(* PLC project PLC1, Beckhoff Automation GmbH TwinCAT PLC Control 3.5.13.21 *)
(* stored: creationDateTime 2023-10-09T14:50:05.3128297, modificationDateTime 2023-10-09T14:50:05.3189547 *)

PROGRAM MAIN
VAR	
	{region 'NC Variables'}
	// Status Array of MCS Position
	MCS_Positions : ARRAY[1..MAX_MCS_AXES] OF LREAL;	
	// Axis Control Ref for ACS
	ACS_Axis		: ARRAY[1..MAX_ACS_AXES] OF Axis_Ref;
	// Axis Control Ref for MCS
	MCS_Axis		: ARRAY[1..MAX_MCS_AXES] OF Axis_Ref;
	// ACS Axis Power Block
	mcACS_Power 	: ARRAY[1..MAX_ACS_AXES] OF MC_Power;
	// MCS Axis Power Block
	mcMCS_Power 	: ARRAY[1..MAX_MCS_AXES] OF MC_Power;
	// Axis Set Position Block
	mcSetPosition 	: ARRAY[1..MAX_ACS_AXES] OF MC_SetPosition;
	{endregion}
		 
	{region  'Kinematics Variables'}
	// Kinematic Model Reference
	{attribute 'TcInitSymbol'}
	oidTrafo			: OTCID;
	// Struct In from Kin Channel
	in_stKinToPlc      AT %I*     : NCTOPLC_NCICHANNEL_REF;
	// Struct Out to Kin Channel
	out_stPlcToKin     AT %Q*     : PLCTONC_NCICHANNEL_REF;	 
	// Axes Configuration Structure
	stAxesConfig		: ST_KinAxes;
	// Kinematics Configuration Group			  
	fbConfigKinGroup	: FB_KinConfigGroup;
	// Reset the Kin Group
	fbResetKinGroup   : FB_KinResetGroup;
	// Calculating the Trafo
	fbKinCalcTrafo		: FB_KinCalcTrafo;
	// Struct of position into the calculation
    stAxesPosIn			: ARRAY[1..8] OF LREAL;
	// Struct of positions out
    stAxesPosOut		: ARRAY[1..8] OF LREAL;			  
	// Scara Meta Info 
	uScaraMetaInfoIn	: U_KinMetaInfo;
	// Scara Meta Info
    uScaraMetaInfoOut	: U_KinMetaInfo;
  	// Unlock Trafo
	fbUnlockTrafoParam	: FB_KinUnlockTrafoParam;
	// Lock Trafo
	fbLockTrafoParam	: FB_KinLockTrafoParam;
	// ADS Write Block
    fbADSWRITE			: ADSWRITE;	
	// Parameter ID to Change (*Inner Arm Length*)
	pidTrafo			: UDINT := 16#05010020; 
	// Value to write to the parameter
	fParamValue			: LREAL := 400.0;			  
	{endregion}

	{region  'General System Variables'}
	// Loop Iterator
	I_itr			: INT;
	{endregion}
		 
	{region 'State Machine Variables'}
	// State of the state machine
	nState 			: INT;
	// Control Variables
	bStart, bHalt, bDoneMoving, bCalcTrafo, bAdjustTrafo, bRepeat : BOOL;
	{endregion}
END_VAR
VAR CONSTANT
	{region  'Axes Constants'}
	// ACS Axes Count
	MAX_ACS_AXES 		: INT := 4;
	// MCS Axes Count
	MAX_MCS_AXES 		: INT := 4;
	// Joint Positions
	AXES_JOINT_POSE	: ARRAY[1..MAX_ACS_AXES] OF LREAL := [0.0, 90.0, 0.0, 0.0];
	{endregion}
END_VAR

            // Simple NC State Machine

CASE nState OF
	0:	// Start the state machine
		IF bStart THEN
			bStart := FALSE;
			nState := nState + 10;
		END_IF
	
	10..40: 
		// Power on all axis (Both ACS and MCS)
		ACS_MCS_Power();
	  
	50: 
		// Step 1 - Assemble the Axes List Struct
		Step_1_Axes_List();
	 
	60..70:	
		// Step 3 - might have an issue at Step 2, so here is where you'll fix it
		Step_3_Fix_Kin_Config();
			   
	80: 
		//	Step 2 - Configure Kinematic Group
		Step_2_Configure_Kin_Group();
					  
	90: 
		(*
		** Move the robot!
		*)
		(*******************************************)	 
		// Command to move on from this step				   
		IF bDoneMoving THEN
			bDoneMoving := FALSE;
			nState := nState + 10;
		END_IF
		(*******************************************)	
		
	100: 
		// Step 5 - Break the Kinematic Group
		Step_5_Reconfig_Kin_Group(); 				   
		 
	110: 
		// Wait state before adjustment
		IF bAdjustTrafo THEN
			bAdjustTrafo := FALSE;
			nState := nState + 10;
		END_IF
	
	120..140:
		// Step 6 - Unlock Trafo and Modify Params
		Step_6_Adjust_Trafo();	 
		
	150: 
		// Check if repeating state machine
		IF bRepeat THEN
			bRepeat := FALSE;
			nState := 60;
		END_IF		
END_CASE


// Step 4 - Calculate the Transformation
IF bCalcTrafo THEN
	Step_4_Calc_Trafo();
END_IF

	 
          

ACTION Step_1_Axes_List:
                (*

// Assign the ACS Axes
FOR I_itr := 1 TO MAX_ACS_AXES DO
	stAxesConfig.nAxisIdsAcs[I_itr] := ACS_Axis[I_itr].NcToPlc.AxisId;
END_FOR
// Assign the MCS Axes
FOR I_itr := 1 TO MAX_MCS_AXES DO
	stAxesConfig.nAxisIdsMcs[I_itr] := MCS_Axis[I_itr].NcToPlc.AxisId;
END_FOR

*)


nState := nState + 10; 		 
              
END_ACTION

ACTION Step_2_Configure_Kin_Group:
                (*
fbConfigKinGroup(bExecute := TRUE, 
					bCartesianMode := TRUE, 
					stAxesList := stAxesConfig, 
					stKinRefIn := in_stKinToPlc); 
					
(*******************************************)
// If you get an error, think about why it doesnt work
IF fbConfigKinGroup.bDone THEN
	nState := nState + 10;	 
END_IF
*)

// Comment Me
nState := nState + 10;	 
              
END_ACTION

ACTION Step_3_Fix_Kin_Config:
                (*
CASE nState OF
	60:	// Step 2 might have an issue, here is where you'll fix it
		(**********************************************************)
		FOR I_itr := 1 TO MAX_ACS_AXES DO
			mcSetPosition[I_itr](Axis := ACS_Axis[I_itr], Execute := TRUE, Position := AXES_JOINT_POSE[I_itr]);		 
	 	END_FOR
		(**********************************************************)	 
		nState := nState + 10; 
			 
	70: // Check if the command is complete
		(**********************************************************)
		FOR I_itr := 1 TO MAX_ACS_AXES DO
			mcSetPosition[I_itr](Axis := ACS_Axis[I_itr], Execute := FALSE, Position := AXES_JOINT_POSE[I_itr]);		 
	 	END_FOR
		(**********************************************************)	 
		nState := nState + 10;
END_CASE
*)

// Comment Me Out
nState := nState + 10;
              
END_ACTION

ACTION Step_4_Calc_Trafo:
                // Toggle eveything false		 
fbKinCalcTrafo(
	bExecute := FALSE,	
	bForward := FALSE, 
	stAxesPosIn := stAxesPosIn, 
	stAxesPosOut := stAxesPosOut, 
	uMetaInfoIn:= uScaraMetaInfoIn, 
	uMetaInfoOut:= uScaraMetaInfoOut);
	 
// Check if Kinematics is running, if not then calculate the MCS
IF F_KinGetChnOperationState(stKinRefIn := in_stKinToPlc) = E_KinStatus.KinStatus_Ready THEN
	FOR I_itr := 1 TO MAX_MCS_AXES DO
		MCS_Positions[I_itr] := MCS_Axis[I_itr].NcToPlc.ActPos;
	END_FOR		 
ELSE
	// Copy the ACS positions for calculation
	FOR I_itr := 1 TO MAX_MCS_AXES DO
		stAxesPosIn[I_itr] := ACS_Axis[I_itr].NcToPlc.ActPos;
	END_FOR		 
	// Tell the calculation that the SCARA is a Right Arm		  
	uScaraMetaInfoIn.eScara := E_KinMetaInfoScara.scaraRightArm;
	
	// Compute the kinematics
	fbKinCalcTrafo(
		bExecute := TRUE, 
		bForward := TRUE, 
		oidTrafo := oidTrafo, 
		stAxesPosIn := stAxesPosIn, 
		stAxesPosOut := stAxesPosOut, 
		uMetaInfoIn:= uScaraMetaInfoIn, 
		uMetaInfoOut:= uScaraMetaInfoOut); 	
			 
	// Copy the computed values into the MCS_Position array
	FOR I_itr := 1 TO MAX_MCS_AXES DO
		MCS_Positions[I_itr] := stAxesPosOut[I_itr];
	END_FOR		  
 END_IF
              
END_ACTION

ACTION Step_5_Reconfig_Kin_Group:
                (*
fbResetKinGroup(
	bExecute := TRUE, 
	nItpChannelId := in_stKinToPlc.ChnId, 
	stKinRefIn := in_stKinToPlc, 
	stAxesList := stAxesConfig);
		 
IF fbResetKinGroup.bDone THEN
	fbResetKinGroup(bExecute := FALSE, nItpChannelId := in_stKinToPlc.ChnId, stKinRefIn := in_stKinToPlc, stAxesList := stAxesConfig);	 
	nState := nState + 10;	 
END_IF	
*)	 

// Comment Me
nState := nState + 10;	
              
END_ACTION

ACTION Step_6_Adjust_Trafo:
                (*CASE nState OF
	120: (*
		** Step 6 - Unlock Trafo and Modify Params
		*)
		(*******************************************)
		fbUnlockTrafoParam(bExecute := TRUE, oidTrafo := oidTrafo);
		IF fbUnlockTrafoParam.bDone THEN
			fbUnlockTrafoParam(bExecute := FALSE, oidTrafo := oidTrafo);
			nState := nState + 10;	 
		END_IF
		(*******************************************)
			 
	130: // Write the value with ADS
		(*******************************************)
		fbADSWRITE(	NETID:='' ,
					PORT:= AMSPORT_R0_NCSAF,
					IDXGRP:=oidTrafo ,
					IDXOFFS:= pidTrafo,
					LEN:=SIZEOF(fParamValue) ,
					SRCADDR:= ADR(fParamValue),
					WRITE:=TRUE);	

		IF NOT fbADSWRITE.BUSY THEN
			fbADSWRITE(WRITE:=FALSE);
			nState := nState + 10;	 
		END_IF	  
		(*******************************************)
	140: // Lock Trafo back up
		(*******************************************)
		fbLockTrafoParam(bExecute := TRUE, oidTrafo := oidTrafo);					   
		IF fbLockTrafoParam.bDone THEN
			fbLockTrafoParam(bExecute := FALSE, oidTrafo := oidTrafo);
			nState := nState + 10;
		END_IF
		(*******************************************)	
END_CASE
*)

// Comment Me
nState := nState + 30;
              
END_ACTION

ACTION ACS_MCS_Power:
                CASE nState OF
	10: // Power on the axis
		FOR I_itr := 1 TO MAX_ACS_AXES DO
			mcACS_Power[I_itr](Axis := ACS_Axis[I_itr], Enable := TRUE, Enable_Positive := TRUE, Enable_Negative := TRUE, Override := 100.0);
		END_FOR
		nState := nState + 10;
	
	20: // Check all axis are enabled
		FOR I_itr := 1 TO MAX_ACS_AXES DO
			// Check if motor is enabled
			IF NOT mcACS_Power[I_itr].Status THEN
				// Return to power state, or reset state if you have one
				// At the end of this state we add 10, so to return to 10 we need to subtract 20
				nState := nState - 20;
				EXIT;
			END_IF
		END_FOR
		nState := nState + 10;

	30: // Power on the axis
		FOR I_itr := 1 TO MAX_MCS_AXES DO
			mcMCS_Power[I_itr](Axis := MCS_Axis[I_itr], Enable := TRUE, Enable_Positive := TRUE, Enable_Negative := TRUE, Override := 100.0);
		END_FOR
		nState := nState + 10;
	
	40: // Check all axis are enabled
		FOR I_itr := 1 TO MAX_MCS_AXES DO
			// Check if motor is enabled
			IF NOT mcMCS_Power[I_itr].Status THEN
				// Return to power state, or reset state if you have one
				// At the end of this state we add 10, so to return to 10 we need to subtract 20
				nState := nState - 20;
				EXIT;
			END_IF
		END_FOR
		nState := nState + 10;
END_CASE
              
END_ACTION
END_PROGRAM
